Fanuc KAREL source: ka00054.KL

-- PROVISIONAL review KL for V770-1; original PC SHA256 cc30cf7bcd6e45868e6161e654a6809e766846bf93e2dd0547bf3a16b3c9be3e
-- Incomplete behavior may be omitted. Consult companion uncertainty JSON. Do not deploy.
PROGRAM KA00054
%NOLOCKGROUP
-- UNRESOLVED_DECL SRC type=000101
-- UNRESOLVED_DECL DST type=000102
BEGIN
  -- UNRESOLVED_PC offsets 5-25; opcodes 49,7E,4A
  -- UNRESOLVED_PC offsets 30-34; opcodes 7F
END KA00054
